SUBAPPLICATION Ventilsteuerung_Uebung_039a (* Spiegelabfolge V2 mit Schrittkette *)
  (* Standard: 61499-2 *)
  (* Version 1.0, 2023-10-23, franz *)
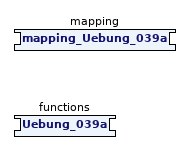
  SUBAPPS
    mapping : mapping_Uebung_039a;
    functions : Uebung_039a;
  END_SUBAPPS
END_SUBAPPLICATION
